PROGRAM PRG_TM1K4
VAR
    {attribute 'pytmc' := '
        pv: TM1K4:ATM
        io: io
    '}
    {attribute 'TcLinkTo' := '.fbThermoCouple1.bError := TIIB[TM1K4-EL3314-E5]^TC Inputs Channel 1^Status^Error;
                              .fbThermoCouple1.bUnderrange := TIIB[TM1K4-EL3314-E5]^TC Inputs Channel 1^Status^Underrange;
                              .fbThermoCouple1.bOverrange := TIIB[TM1K4-EL3314-E5]^TC Inputs Channel 1^Status^Overrange;
                              .fbThermoCouple1.iRaw := TIIB[TM1K4-EL3314-E5]^TC Inputs Channel 1^Value'}
    fbTM1K4: FB_ATM;
END_VAR

fbTM1K4.nTransitionAssertionID := 16#5140;
fbTM1K4.nUnknownAssertionID := 16#5149;

fbTM1K4.stOut.fPosition := -15;
fbTM1K4.stOut.bUseRawCounts := FALSE;
fbTM1K4.stOut.nRequestAssertionID := 16#5141;
fbTM1K4.stOut.stBeamParams := PMPS_GVL.cstFullBeam;
fbTM1K4.stOut.bValid := TRUE;

fbTM1K4.stTarget1.fPosition := -39.124;
fbTM1K4.stTarget1.bUseRawCounts := FALSE;
fbTM1K4.stTarget1.nRequestAssertionID := 16#5142;
fbTM1K4.stTarget1.stBeamParams := PMPS_GVL.cstFullBeam;
fbTM1K4.stTarget1.bValid := TRUE;

fbTM1K4.stTarget2.fPosition := -53.5;
fbTM1K4.stTarget2.bUseRawCounts := FALSE;
fbTM1K4.stTarget2.nRequestAssertionID := 16#5143;
fbTM1K4.stTarget2.stBeamParams := PMPS_GVL.cstFullBeam;
fbTM1K4.stTarget2.bValid := TRUE;

fbTM1K4.stTarget3.fPosition := -67.874;
fbTM1K4.stTarget3.bUseRawCounts := FALSE;
fbTM1K4.stTarget3.nRequestAssertionID := 16#5144;
fbTM1K4.stTarget3.stBeamParams := PMPS_GVL.cstFullBeam;
fbTM1K4.stTarget3.bValid := TRUE;

fbTM1K4.stTarget4.fPosition := -82.25;
fbTM1K4.stTarget4.bUseRawCounts := FALSE;
fbTM1K4.stTarget4.nRequestAssertionID := 16#5145;
fbTM1K4.stTarget4.stBeamParams := PMPS_GVL.cstFullBeam;
fbTM1K4.stTarget4.bValid := TRUE;

fbTM1K4.stTarget5.fPosition := -96.623;
fbTM1K4.stTarget5.bUseRawCounts := FALSE;
fbTM1K4.stTarget5.nRequestAssertionID := 16#5146;
fbTM1K4.stTarget5.stBeamParams := PMPS_GVL.cstFullBeam;
fbTM1K4.stTarget5.bValid := TRUE;

fbTM1K4(
    fbArbiter := fbArbiter,
    fbFFHWO := fbFastFaultOutput1,
    stYStage := Main.M21,
    stXStage := Main.M22);

END_PROGRAM

(* stored: Version 1.1.0.1, ProductVersion 3.1.4022.18
   POU PRG_TM1K4: Id {c02e8350-6bfd-4c3f-8509-cf01c04221fa}, SpecialFunc None *)
